(* CODESYS project CtaSysGrafanaLibPanel_1.0.0.0.library
   Description: SYS Grafana Library der CTA
   Version: 1.0.0.0
   Title: CtaSysGrafanaLibPanel
   Author: SIS
   Company: CTA
   Placeholder: CtaSysGrafanaLibPanel
   DocFormat: reStructuredText
   CompiledLibraryCompatibilityVersion: CODESYS V3.5 SP16 Patch 3
   LanguageModelAttribute: qualified-access-only
   DefaultNamespace: CtaSysGrafanaLibPanel

Project tree, tasks and I/O mapping:
  libraries: SysProcess, 3.5.17.0 (System); Standard, 3.5.18.0 (System); StringUtils, 3.5.18.0 (System); CtaVisSymbols, 1.0.0.0 (CTA); VisuSymbols, 4.5.0.0 (System); SysTypes Interfaces, * (System)
  40 Visualizations/
    visualisation VIS_GRAFANA_LIB_PANEL
    visualisation VIS_POPUP_GRAFANA
  00000000-0000-0000-0000-000000000000|D:\CoDeSys\LibrariesV3\trunk\Intern\CAA\CAA Template\3.4.0.0 draft\Placeholder.xml
  00000000-0000-0000-0000-000000000000|D:\CoDeSys\LibrariesV3\trunk\Intern\CAA\CAA Template\3.2.0.3 draft\Prefix.pdf
  00000000-0000-0000-0000-000000000000|D:\CoDeSys\LibrariesV3\trunk\Intern\CAA\CAA Template\3.5.2.0 draft\Placeholder.xml
  20 Structs/
  50 Images/
  10 Documenation/
    global variables VersionHistory
    global variables readMe
  21 Interface/
    interface ITF_GRAFANA_LIB_PANEL: TABLE_EXECUTE, TABLE_STATUS, LIB_PANEL_UID
  11 Library Parameter/
    global variables Parameter
  12 Konstanten/
  60 Textlisten/
  13 Globale Variablen/
    global variables GVL_GRAFANA_CONSTANT
    global variables GVL_GRAFANA_LIB_PANEL
  text list GlobalTextList
  5ce3da45-db07-42e7-a21c-a00fff4ed8f6|C:\Users\sis\Downloads\dip-switch.svg
  5ce3da45-db07-42e7-a21c-a00fff4ed8f6|C:\Users\sis\Downloads\lightning-bolt-circle.svg
  30 Program Organization Units/
    function block FB_GRAFANA_LIB_PANEL [ST]: TIMESERIES_HEAD, TIMESERIES_FOOTER, STATETIMELINE_HEAD, STATETIMELINE_FOOTER, GET_VERSION, UPDATE_VERSION, DO_HEADER, DO_FOOTER, DO_TEMP_FILES, DELETE_TEMP_FILES, URL, NEW_LIB_PANEL, UPDATE_LIB_PANEL, GET_LIB_PANEL, GET_API_KEY, DELETE_API_KEY, DATA, READY_FOR_DATA, FB_EXIT, FB_INIT, TABLE_STATUS, EXECUTE, LIB_PANEL_UID, TABLE_EXECUTE, REMOVE_SPECIALCHAR, CREATE_DYN_DATA, DELETE_DYN_DATA
    function fcRemoveSpezialChar [ST]
  5ce3da45-db07-42e7-a21c-a00fff4ed8f6|C:\Users\sis\Downloads\sine-wave.svg
  5ce3da45-db07-42e7-a21c-a00fff4ed8f6|C:\Users\sis\Downloads\eye.svg
  5ce3da45-db07-42e7-a21c-a00fff4ed8f6|C:\Users\sis\Downloads\lan.svg
  22 Enumeration/
    data type FB_GRAFANA_LIB_PANEL_STATUS
    data type GRAFANA_DATABASE_TYPE
    data type GRAFANA_LIB_PANEL_TYPE
*)

// 22 Enumeration/FB_GRAFANA_LIB_PANEL_STATUS
{attribute 'qualified_only'}
{attribute 'strict'}
TYPE FB_GRAFANA_LIB_PANEL_STATUS :
(
	NO_ERROR		:= -1,
	READY 			:= 0,
	GET_API_KEY		:= 1,
	DO_TMP_FILE		:= 2,
	DO_JSON_HEADER	:= 3,
	DO_JSON_DATA	:= 4,
	DO_JSON_FOOTER	:= 5,
	DO_NEW_PANEL	:= 6,
	DO_UPDATE		:= 7,
	DELETE_API_KEY	:= 8,
	DELETE_DYNMEM	:= 9
);
END_TYPE

// 22 Enumeration/GRAFANA_DATABASE_TYPE
{attribute 'qualified_only'}
{attribute 'strict'}
TYPE GRAFANA_DATABASE_TYPE :
(
	INFLUXDB := 1
);
END_TYPE

// 22 Enumeration/GRAFANA_LIB_PANEL_TYPE
{attribute 'qualified_only'}
{attribute 'strict'}
TYPE GRAFANA_LIB_PANEL_TYPE :
(
	TIMESERIES 		:= 0,
	STATETIMELINE 	:= 1
);
END_TYPE

// 10 Documenation/VersionHistory
(* 

.. image:: ../../Images/CTA_Logo.jpg
   :align: right
   :width: 15% 

**Vorlage**   


============ =========== =========== ============================================
**Date**     **Version** **Author**  **Change**
------------ ----------- ----------- --------------------------------------------
04.03.2021   0.0.0.0     SIS         Vorlage erstellt

============ =========== =========== ============================================


*)
VAR_GLOBAL
    stInfo : STRING:= '0.0.0.0, Vorlage, CTA';
END_VAR

// 10 Documenation/readMe
(*

**ReadMe**
 
|	**Empfehlung**
|
|	Die SysGrafanaLibPanel Library dient der automatischen erstellung von Grafana Library Panels. Diese können mit dem FB_GRAFANA_LIB_PANEL erstellt werden.
|	Die erstellung des Panels wird Manuell über die Visualisierung ausgelöst. 
|	Die Daten welche für das erstellen der Panel benötigt werden können über die Methode DATA abgefüllt werden. Jeder Aufruf der Methode ist ein Data field.
|  
| *Beispiel* 

+-----------------------+---------------------------------------------------------------------------------------------------------------------------------------------------------------------------------------------------------------------------------------------------------------------------------------------------------------------------------------------------------------------------------------------------------------------------------------+
| Beschreibung          |  Code                                                                                                                                                                                                                                                                                                                                                                                                                                 |
+=======================+=======================================================================================================================================================================================================================================================================================================================================================================================================================================+
| Pou oder SmFb         | .. code-block:: codesys                                                                                                                                                                                                                                                                                                                                                                                                               |
|                       |                                                                                                                                                                                                                                                                                                                                                                                                                                       |
|                       |	// Deklaration als VAR im POU oder dem selbsterstellten Funktionsbaustein                                                                                                                                                                                                                                                                                                                                                       	|
|                       |   VAR   																																																																																																								|
|						|	    (*Grafana Test Panel*)																																																		 																																																	|
|						|		fbGrafanaTestPanel  : CtaSysGrafanaLibPanel.FB_GRAFANA_LIB_PANEL;                                                                                                                                                                                                                                                                                                                                								|
| 						|	END_VAR                                                                                                                                                                                                                                                                                                                                                                                                                         	|
+-----------------------+---------------------------------------------------------------------------------------------------------------------------------------------------------------------------------------------------------------------------------------------------------------------------------------------------------------------------------------------------------------------------------------------------------------------------------------+
| Code                  | .. code-block:: codesys                                                                                                                                                                                                                                                                                                                                                                                                               |
|                       |   																																																																																																									|
| 						|																																																																																																										|
|                       |	fbGrafanaTestPanel(	LIB_PANEL_TYPE	:= GRAFANA_LIB_PANEL_TYPE.TIMESERIES,																																																																																							|
| 						|						DATABASE_TYPE	:= GRAFANA_DATABASE_TYPE.INFLUXDB,               																																																																																				|
|						|						stDATABASE_NAME	:= CtaAppTrendLog.fcGetInfluxDbName,	                             																																																																															|
|						|						stLIB_PANEL_UID := "UniqPanelName",                         																																																																																					| 
|						|						stIP			:= CtaAppTrendLog.fcGetInfluxDbIp,                                         																																																																														| 
|						|						uiPORT			:= CtaAppTrendLog.fcGetInfluxDbPort,                                              																																																																												| 
|						|						stUSER			:= 'admin',                                           																																																																																			|
|						|						stPASSWORD		:= 'CtaElektro');                                  																																																																																				| 
|						|																																																																																																										| 
|						|																										   	 																																																																															| 
|						|	IF fbGrafanaTestPanel.READY_FOR_DATA() THEN																											    																																																																			| 
|						|		fbGrafanaTestPanel.DATA("TrendLogId","Alias","BOOL?","LetztesFeld?");                       																																				    																																												| 
|						|	END_IF;																																													    																																																										| 
|						|																				    																																																																																					| 
|						|																																					    																																																																				| 
|						|																																																																																																										| 
|						|																																																																																																										| 
|						|																																																																																																										| 
+-----------------------+---------------------------------------------------------------------------------------------------------------------------------------------------------------------------------------------------------------------------------------------------------------------------------------------------------------------------------------------------------------------------------------------------------------------------------------+
*)      
VAR_GLOBAL
    xReadMeDone              :   BOOL;
END_VAR

// 13 Globale Variablen/GVL_GRAFANA_CONSTANT
{attribute 'qualified_only'}
VAR_GLOBAL CONSTANT
	MAX_SUPORTET_DATABASES	 : INT	:= 1;
	AY_GRAFANA_DATABASE_TYPE : ARRAY[1..MAX_SUPORTET_DATABASES] OF STRING	:= ['influxdb'];
END_VAR

// 13 Globale Variablen/GVL_GRAFANA_LIB_PANEL
{attribute 'qualified_only'}
VAR_GLOBAL
	AY_FB_GRAFANA_LIB_PANEL	:	ARRAY[1..Parameter.iMaxLibPanels] OF ITF_GRAFANA_LIB_PANEL;
	diMissedMemory			:	DINT;
	diNextFreePlace			:	DINT;
	iMaxShow				:	INT;
	xMemoryError			:	BOOL;
	dwSync					:	DWORD;
END_VAR

// 11 Library Parameter/Parameter
{attribute 'qualified_only'}
VAR_GLOBAL CONSTANT
    iMaxLibPanels :   INT   := 60;         // Maximale Anzahl verwendeter AT-Bausteine    
END_VAR

// 30 Program Organization Units/FB_GRAFANA_LIB_PANEL
FUNCTION_BLOCK FB_GRAFANA_LIB_PANEL IMPLEMENTS ITF_GRAFANA_LIB_PANEL
VAR_INPUT
	LIB_PANEL_TYPE	:	GRAFANA_LIB_PANEL_TYPE;
	DATABASE_TYPE	:	GRAFANA_DATABASE_TYPE;
	stDATABASE_NAME	:	STRING(40);
	stLIB_PANEL_UID	:	STRING(40);
	stIP			:	STRING(15);
	uiPORT			:	UINT;
	stUSER			:	STRING;
	stPASSWORD		:	STRING;
END_VAR
VAR_OUTPUT
	xREADY			:	BOOL;
	xBUSY			:	BOOL;
	xOK				:	BOOL	:= TRUE;
	xERROR			:	BOOL;
	ERROR_ON_STATE	:	FB_GRAFANA_LIB_PANEL_STATUS;	
END_VAR
VAR
	stLIB_PANEL_UID_NO_SPC	:	STRING;
	xExecute				:	BOOL;
	stURL					:	POINTER TO STRING(255);
	stKEY					:	POINTER TO STRING(255);
	stKEY_ID				:	POINTER TO STRING(10);
	stVersion				:	POINTER TO STRING(40);
	stResult				:	POINTER TO STRING(255);	
	stTemp					:	POINTER TO STRING(2000);
	stCommand				:	POINTER TO STRING(2000);
	RTS_IEC_RESULT			:	SysTypes.RTS_IEC_RESULT;
	STATUS					:	FB_GRAFANA_LIB_PANEL_STATUS;
	uiDataSecurity			:	UINT;
	dwTest					:	DWORD;
END_VAR

(* STATE MACHINE *)
CASE STATUS OF
	(* READY *)
	FB_GRAFANA_LIB_PANEL_STATUS.READY 			:
		xREADY	:= TRUE;
		xBUSY	:= FALSE;
		IF xExecute THEN
			xREADY			:= FALSE;
			xBUSY			:= TRUE;
			dwTest := TEST_AND_SET(GVL_GRAFANA_LIB_PANEL.dwSync);
			IF dwTest = 0 THEN
				CREATE_DYN_DATA();
				URL();	
				STATUS 			:= FB_GRAFANA_LIB_PANEL_STATUS.GET_API_KEY;					
				ERROR_ON_STATE	:= FB_GRAFANA_LIB_PANEL_STATUS.NO_ERROR;
				xOK    			:= FALSE;
				xERROR 			:= FALSE;
				xExecute		:= FALSE;
				uiDataSecurity	:= 0;
			END_IF;
		END_IF;	
	
	(* GET API KEY *)
	FB_GRAFANA_LIB_PANEL_STATUS.GET_API_KEY		:
		REMOVE_SPECIALCHAR();
		GET_API_KEY();
		IF xERROR AND ERROR_ON_STATE = FB_GRAFANA_LIB_PANEL_STATUS.NO_ERROR THEN
			ERROR_ON_STATE := FB_GRAFANA_LIB_PANEL_STATUS.GET_API_KEY;
		END_IF;
		
	(* DO TEMP FILE *)
	FB_GRAFANA_LIB_PANEL_STATUS.DO_TMP_FILE		:
		DO_TEMP_FILES();
		IF xERROR AND ERROR_ON_STATE = FB_GRAFANA_LIB_PANEL_STATUS.NO_ERROR THEN
			ERROR_ON_STATE := FB_GRAFANA_LIB_PANEL_STATUS.DO_TMP_FILE;
		END_IF;
		
	(* DO JSON HEADER *)
	FB_GRAFANA_LIB_PANEL_STATUS.DO_JSON_HEADER	:
		DO_HEADER();
		IF xERROR AND ERROR_ON_STATE = FB_GRAFANA_LIB_PANEL_STATUS.NO_ERROR THEN
			ERROR_ON_STATE := FB_GRAFANA_LIB_PANEL_STATUS.DO_JSON_HEADER;
		END_IF;
		
	(* DO JSON DATA *)
	FB_GRAFANA_LIB_PANEL_STATUS.DO_JSON_DATA		:
		(* Wait for DATA *) ;
		IF xERROR AND ERROR_ON_STATE = FB_GRAFANA_LIB_PANEL_STATUS.NO_ERROR THEN
			ERROR_ON_STATE := FB_GRAFANA_LIB_PANEL_STATUS.DO_JSON_DATA;
		END_IF;	
		
	(* DO JSON FOOTER *)	
	FB_GRAFANA_LIB_PANEL_STATUS.DO_JSON_FOOTER	:
		DO_FOOTER();
		IF xERROR AND ERROR_ON_STATE = FB_GRAFANA_LIB_PANEL_STATUS.NO_ERROR THEN
			ERROR_ON_STATE := FB_GRAFANA_LIB_PANEL_STATUS.DO_JSON_FOOTER;
		END_IF;
		
	(* DO NEW PANEL *)
	FB_GRAFANA_LIB_PANEL_STATUS.DO_NEW_PANEL		:
		NEW_LIB_PANEL();
		IF xERROR AND ERROR_ON_STATE = FB_GRAFANA_LIB_PANEL_STATUS.NO_ERROR THEN
			ERROR_ON_STATE := FB_GRAFANA_LIB_PANEL_STATUS.DO_NEW_PANEL;
		END_IF;
		
	(* DO PANEL UPDATE *)
	FB_GRAFANA_LIB_PANEL_STATUS.DO_UPDATE		:
		UPDATE_LIB_PANEL();
		IF xERROR AND ERROR_ON_STATE = FB_GRAFANA_LIB_PANEL_STATUS.NO_ERROR THEN
			ERROR_ON_STATE := FB_GRAFANA_LIB_PANEL_STATUS.DO_UPDATE;
		END_IF;
		
	(* DELETE API KEY *)
	FB_GRAFANA_LIB_PANEL_STATUS.DELETE_API_KEY	:
		DELETE_API_KEY();
		DELETE_TEMP_FILES();
		xOK 	:= NOT xERROR;
		STATUS	:= FB_GRAFANA_LIB_PANEL_STATUS.DELETE_DYNMEM;
		IF xERROR AND ERROR_ON_STATE = FB_GRAFANA_LIB_PANEL_STATUS.NO_ERROR THEN
			ERROR_ON_STATE := FB_GRAFANA_LIB_PANEL_STATUS.DELETE_API_KEY;
		END_IF;
	(* DELETE MEM *)
	FB_GRAFANA_LIB_PANEL_STATUS.DELETE_DYNMEM :
		DELETE_DYN_DATA();
		STATUS	:= FB_GRAFANA_LIB_PANEL_STATUS.READY;
		GVL_GRAFANA_LIB_PANEL.dwSync := 0;
	ELSE
		STATUS := FB_GRAFANA_LIB_PANEL_STATUS.DELETE_DYNMEM;
END_CASE

METHOD PRIVATE TIMESERIES_HEAD : BOOL
VAR_INPUT
END_VAR
IF stURL <> 0 AND stKEY <> 0 AND stKEY_ID <> 0 AND stVersion <> 0 AND stResult <> 0 AND stTemp <> 0 AND stCommand <> 0 THEN
	stCommand^ := '';
	stTemp^:= '';
	stTemp^:= 'echo $'{
	"uid": "';
	Stu.StrConcatA(pstFrom:= ADR(stTemp^),pstTo := ADR(stCommand^),TO_INT(SIZEOF(stCommand^)));
	stTemp^:= '';
	stTemp^:= stLIB_PANEL_UID_NO_SPC;
	Stu.StrConcatA(pstFrom:= ADR(stTemp^),pstTo := ADR(stCommand^),TO_INT(SIZEOF(stCommand^)));
	stTemp^ := '';
	stTemp^ := '",
	"folderId": 0,
	"name": "';
	Stu.StrConcatA(pstFrom:= ADR(stTemp^),pstTo := ADR(stCommand^),TO_INT(SIZEOF(stCommand^)));
	stTemp^:= '';
	stTemp^:= stLIB_PANEL_UID;
	Stu.StrConcatA(pstFrom:= ADR(stTemp^),pstTo := ADR(stCommand^),TO_INT(SIZEOF(stCommand^)));
	stTemp^ := '';
	stTemp^ := '",
	  "version": 1,
	  "model":
	{
	  "type": "timeseries",
	  "title": "';
	Stu.StrConcatA(pstFrom:= ADR(stTemp^),pstTo := ADR(stCommand^),TO_INT(SIZEOF(stCommand^)));
	stTemp^ := '';
	stTemp^ := stLIB_PANEL_UID;
	Stu.StrConcatA(pstFrom:= ADR(stTemp^),pstTo := ADR(stCommand^),TO_INT(SIZEOF(stCommand^)));
	stTemp^ := '';
	stTemp^ := '",
		"targets": [
		{
		  "refId": "A",
		  "datasource": {
			"type": "';
	Stu.StrConcatA(pstFrom:= ADR(stTemp^),pstTo := ADR(stCommand^),TO_INT(SIZEOF(stCommand^)));
	
	stTemp^ := '';
	IF DATABASE_TYPE >= GRAFANA_DATABASE_TYPE.INFLUXDB AND DATABASE_TYPE <= GVL_GRAFANA_CONSTANT.MAX_SUPORTET_DATABASES THEN
		stTemp^ := GVL_GRAFANA_CONSTANT.AY_GRAFANA_DATABASE_TYPE[DATABASE_TYPE];
	ELSE
		stTemp^ := GVL_GRAFANA_CONSTANT.AY_GRAFANA_DATABASE_TYPE[GRAFANA_DATABASE_TYPE.INFLUXDB];	
	END_IF;
	Stu.StrConcatA(pstFrom:= ADR(stTemp^),pstTo := ADR(stCommand^),TO_INT(SIZEOF(stCommand^)));
	
	stTemp^ := '';
	stTemp^ := '",
			"uid": ""
		  },
		  "policy": "default",
		  "resultFormat": "time_series",
		  "orderByTime": "ASC",
		  "tags": [],
		  "groupBy": [
			{
			  "type": "time",
			  "params": [
				"$$__interval"
			  ]
			},
			{
			  "type": "fill",
			  "params": [
				"none"
			  ]
			}
		  ],
		  "select": [$' > /tmp/';
	Stu.StrConcatA(pstFrom:= ADR(stTemp^),pstTo := ADR(stCommand^),TO_INT(SIZEOF(stCommand^)));
	stTemp^ := '';
	stTemp^ := stLIB_PANEL_UID_NO_SPC;
	
	Stu.StrConcatA(pstFrom:= ADR(stTemp^),pstTo := ADR(stCommand^),TO_INT(SIZEOF(stCommand^)));
	stTemp^ := '';
	stTemp^ := '.txt';
	Stu.StrConcatA(pstFrom:= ADR(stTemp^),pstTo := ADR(stCommand^),TO_INT(SIZEOF(stCommand^)));
		  
	SysProcess_Implementation.SysProcessExecuteCommand2(stCommand^,stResult^,SIZEOF(stResult^),ADR(RTS_IEC_RESULT));
	
	TIMESERIES_HEAD	:= RTS_IEC_RESULT = 0;
ELSE
	STATUS := FB_GRAFANA_LIB_PANEL_STATUS.DELETE_DYNMEM;
END_IF;
END_METHOD

METHOD PRIVATE TIMESERIES_FOOTER : BOOL;
VAR_INPUT
END_VAR
IF stURL <> 0 AND stKEY <> 0 AND stKEY_ID <> 0 AND stVersion <> 0 AND stResult <> 0 AND stTemp <> 0 AND stCommand <> 0 THEN
	stCommand^ := '';
	stCommand^ := 'echo $'],
				  "measurement": "';
	stTemp^ := '';
	stTemp^ := stDATABASE_NAME;
	
	Stu.StrConcatA(pstFrom:= ADR(stTemp^),pstTo := ADR(stCommand^),TO_INT(SIZEOF(stCommand^)));
	
	stTemp^ := '';
	stTemp^ := '",
				  "alias": "$$col"
					}
					  ],
					  "options": {
						"tooltip": {
						  "mode": "multi"
						},
						"legend": {
						  "displayMode": "table",
						  "placement": "bottom",
						  "calcs": []
						}
					  },
					  "fieldConfig": {
						"defaults": {
						  "custom": {
							"drawStyle": "line",
							"lineInterpolation": "smooth",
							"barAlignment": 0,
							"lineWidth": 1,
							"fillOpacity": 0,
							"gradientMode": "none",
							"spanNulls": false,
							"showPoints": "auto",
							"pointSize": 5,
							"stacking": {
							  "mode": "none",
							  "group": "A"
							},
							"axisPlacement": "auto",
							"axisLabel": "",
							"scaleDistribution": {
							  "type": "linear"
							},
							"hideFrom": {
							  "tooltip": false,
							  "viz": false,
							  "legend": false
							},
							"thresholdsStyle": {
							  "mode": "off"
							}
						  },
						  "color": {
							"mode": "palette-classic"
						  },
						  "thresholds": {
							"mode": "absolute",
							"steps": [
							  {
								"color": "green",
								"value": null
							  }
							]
						  },
						  "mappings": []
						},
						"overrides": []
					  },
					  "datasource": null
					},
			  "kind": 1
			}$' >> /tmp/';
	Stu.StrConcatA(pstFrom:= ADR(stTemp^),pstTo := ADR(stCommand^),TO_INT(SIZEOF(stCommand^)));
	
	stTemp^ := '';
	stTemp^ := stLIB_PANEL_UID_NO_SPC;
	
	Stu.StrConcatA(pstFrom:= ADR(stTemp^),pstTo := ADR(stCommand^),TO_INT(SIZEOF(stCommand^)));
	stTemp^ := '';
	stTemp^ := '.txt';		
	Stu.StrConcatA(pstFrom:= ADR(stTemp^),pstTo := ADR(stCommand^),TO_INT(SIZEOF(stCommand^)));
	
	SysProcess_Implementation.SysProcessExecuteCommand2(stCommand^,stResult^,SIZEOF(stResult^),ADR(RTS_IEC_RESULT));
	
	TIMESERIES_FOOTER	:= RTS_IEC_RESULT = 0;
ELSE
	STATUS := FB_GRAFANA_LIB_PANEL_STATUS.DELETE_DYNMEM;
END_IF;
END_METHOD

METHOD PRIVATE STATETIMELINE_HEAD : BOOL
VAR_INPUT
END_VAR
IF stURL <> 0 AND stKEY <> 0 AND stKEY_ID <> 0 AND stVersion <> 0 AND stResult <> 0 AND stTemp <> 0 AND stCommand <> 0 THEN
	stCommand^ := '';
	stTemp^:= '';
	stTemp^:= 'echo $'{
	"uid": "';
	Stu.StrConcatA(pstFrom:= ADR(stTemp^),pstTo := ADR(stCommand^),TO_INT(SIZEOF(stCommand^)));
	stTemp^:= '';
	stTemp^:= stLIB_PANEL_UID_NO_SPC;
	Stu.StrConcatA(pstFrom:= ADR(stTemp^),pstTo := ADR(stCommand^),TO_INT(SIZEOF(stCommand^)));
	stTemp^ := '';
	stTemp^ := '",
	"folderId": 0,
	"name": "';
	Stu.StrConcatA(pstFrom:= ADR(stTemp^),pstTo := ADR(stCommand^),TO_INT(SIZEOF(stCommand^)));
	stTemp^:= '';
	stTemp^:= stLIB_PANEL_UID;
	Stu.StrConcatA(pstFrom:= ADR(stTemp^),pstTo := ADR(stCommand^),TO_INT(SIZEOF(stCommand^)));
	stTemp^ := '';
	stTemp^ := '",
	  "version": 1,
	  "model":
	{
	  "type": "state-timeline",
	  "title": "';
	Stu.StrConcatA(pstFrom:= ADR(stTemp^),pstTo := ADR(stCommand^),TO_INT(SIZEOF(stCommand^)));
	stTemp^ := '';
	stTemp^ := stLIB_PANEL_UID;
	Stu.StrConcatA(pstFrom:= ADR(stTemp^),pstTo := ADR(stCommand^),TO_INT(SIZEOF(stCommand^)));
	stTemp^ := '';
	stTemp^ := '",
	  "fieldConfig": {
		"defaults": {
		  "custom": {
			"lineWidth": 0,
			"fillOpacity": 70
		  },
		  "color": {
			"mode": "fixed"
		  },
		  "thresholds": {
			"mode": "absolute",
			"steps": [
			  {
				"color": "green",
				"value": null
			  }
			]
		  },
		  "mappings": []
		},
		"overrides": []
	  },
	  "options": {
		"mergeValues": true,
		"showValue": "auto",
		"alignValue": "left",
		"rowHeight": 0.9,
		"legend": {
		  "displayMode": "hidden",
		  "placement": "bottom"
		},
		"tooltip": {
		  "mode": "single"
		}
	  },
	  "targets": [
		{
		  "datasource": {
			"type": "';
	
	Stu.StrConcatA(pstFrom:= ADR(stTemp^),pstTo := ADR(stCommand^),TO_INT(SIZEOF(stCommand^)));
			
	stTemp^ := '';
	IF DATABASE_TYPE >= GRAFANA_DATABASE_TYPE.INFLUXDB AND DATABASE_TYPE <= GVL_GRAFANA_CONSTANT.MAX_SUPORTET_DATABASES THEN
		stTemp^ := GVL_GRAFANA_CONSTANT.AY_GRAFANA_DATABASE_TYPE[DATABASE_TYPE];
	ELSE
		stTemp^ := GVL_GRAFANA_CONSTANT.AY_GRAFANA_DATABASE_TYPE[GRAFANA_DATABASE_TYPE.INFLUXDB];	
	END_IF;
	Stu.StrConcatA(pstFrom:= ADR(stTemp^),pstTo := ADR(stCommand^),TO_INT(SIZEOF(stCommand^)));
	
	stTemp^ := '';
	stTemp^ := '",
			"uid": ""
		  },
		  "groupBy": [
			{
			  "params": [
				"$$__interval"
			  ],
			  "type": "time"
			},
			{
			  "params": [
				"none"
			  ],
			  "type": "fill"
			}
		  ],
		  "measurement": "';
	
	Stu.StrConcatA(pstFrom:= ADR(stTemp^),pstTo := ADR(stCommand^),TO_INT(SIZEOF(stCommand^)));
	
	stTemp^ := '';
	stTemp^ := stDATABASE_NAME;
	
	Stu.StrConcatA(pstFrom:= ADR(stTemp^),pstTo := ADR(stCommand^),TO_INT(SIZEOF(stCommand^)));
	
	stTemp^ := '';
	stTemp^ := '",
		  "orderByTime": "ASC",
		  "policy": "default",
		  "refId": "A",
		  "resultFormat": "time_series",
		  "select": [$' > /tmp/';
	Stu.StrConcatA(pstFrom:= ADR(stTemp^),pstTo := ADR(stCommand^),TO_INT(SIZEOF(stCommand^)));
	stTemp^ := '';
	stTemp^ := stLIB_PANEL_UID_NO_SPC;
	
	Stu.StrConcatA(pstFrom:= ADR(stTemp^),pstTo := ADR(stCommand^),TO_INT(SIZEOF(stCommand^)));
	stTemp^ := '';
	stTemp^ := '.txt';
	Stu.StrConcatA(pstFrom:= ADR(stTemp^),pstTo := ADR(stCommand^),TO_INT(SIZEOF(stCommand^)));
		  
	SysProcess_Implementation.SysProcessExecuteCommand2(stCommand^,stResult^,SIZEOF(stResult^),ADR(RTS_IEC_RESULT));
	
	STATETIMELINE_HEAD	:= RTS_IEC_RESULT = 0;
ELSE
	STATUS := FB_GRAFANA_LIB_PANEL_STATUS.DELETE_DYNMEM;
END_IF;
END_METHOD

METHOD PRIVATE STATETIMELINE_FOOTER : BOOL
VAR_INPUT
END_VAR
IF stURL <> 0 AND stKEY <> 0 AND stKEY_ID <> 0 AND stVersion <> 0 AND stResult <> 0 AND stTemp <> 0 AND stCommand <> 0 THEN
	stCommand^ := '';
	stCommand^ := 'echo $'],
				  "tags": [],
				  "alias": "$$col"
				}
			  ],
			  "id": 0,
			  "datasource": null
			},
			  "kind": 1
			}$' >> /tmp/';
	
	stTemp^ := '';
	stTemp^ := stLIB_PANEL_UID_NO_SPC;
	
	Stu.StrConcatA(pstFrom:= ADR(stTemp^),pstTo := ADR(stCommand^),TO_INT(SIZEOF(stCommand^)));
	stTemp^ := '';
	stTemp^ := '.txt';		
	Stu.StrConcatA(pstFrom:= ADR(stTemp^),pstTo := ADR(stCommand^),TO_INT(SIZEOF(stCommand^)));
	
	SysProcess_Implementation.SysProcessExecuteCommand2(stCommand^,stResult^,SIZEOF(stResult^),ADR(RTS_IEC_RESULT));
	
	STATETIMELINE_FOOTER	:= RTS_IEC_RESULT = 0;
ELSE
	STATUS := FB_GRAFANA_LIB_PANEL_STATUS.DELETE_DYNMEM;
END_IF;
END_METHOD

METHOD PRIVATE GET_VERSION : BOOL
VAR_INPUT
END_VAR
IF stURL <> 0 AND stKEY <> 0 AND stKEY_ID <> 0 AND stVersion <> 0 AND stResult <> 0 AND stTemp <> 0 AND stCommand <> 0 THEN
	(* Get Version *)
	stCommand^ := '';
	stCommand^ := Standard.CONCAT(Standard.CONCAT('grep -oE $'.{0,1}version.{0,5}[0-9]$' /tmp/',stLIB_PANEL_UID_NO_SPC),'_V.txt | tail -1');
	SysProcess_Implementation.SysProcessExecuteCommand2(stCommand^,stResult^,SIZEOF(stResult^),ADR(RTS_IEC_RESULT));
	
	IF FIND(stResult^,'$N') > 1 AND FIND(stResult^,'"version"') > 0 AND RTS_IEC_RESULT = 0 THEN
		stVersion^ 	:= '';
		stVersion^ 	:= Standard.LEFT(stResult^,FIND(stResult^,'$N')-1);
		GET_VERSION := TRUE;
	ELSE
		xERROR		:= TRUE;
	END_IF;
ELSE
	STATUS := FB_GRAFANA_LIB_PANEL_STATUS.DELETE_DYNMEM;
END_IF;
END_METHOD

METHOD PRIVATE UPDATE_VERSION : BOOL
VAR_INPUT
END_VAR
IF stURL <> 0 AND stKEY <> 0 AND stKEY_ID <> 0 AND stVersion <> 0 AND stResult <> 0 AND stTemp <> 0 AND stCommand <> 0 THEN
	(* Update Version *)
	stCommand^ := '';
	stCommand^ := Standard.CONCAT(Standard.CONCAT(Standard.CONCAT(Standard.CONCAT('sed -i $'s/"version": 1/',stVersion^),'/$' /tmp/'),stLIB_PANEL_UID_NO_SPC),'.txt');
	SysProcess_Implementation.SysProcessExecuteCommand2(stCommand^,stResult^,SIZEOF(stResult),ADR(RTS_IEC_RESULT));
	
	UPDATE_VERSION := RTS_IEC_RESULT = 0;
ELSE
	STATUS := FB_GRAFANA_LIB_PANEL_STATUS.DELETE_DYNMEM;
END_IF;
END_METHOD

METHOD PRIVATE DO_HEADER : BOOL
VAR_INPUT
END_VAR
IF LIB_PANEL_TYPE = GRAFANA_LIB_PANEL_TYPE.TIMESERIES THEN
	IF TIMESERIES_HEAD()	THEN
		STATUS := FB_GRAFANA_LIB_PANEL_STATUS.DO_JSON_DATA;
	ELSE
		STATUS 	:= FB_GRAFANA_LIB_PANEL_STATUS.DELETE_API_KEY;
		xERROR	:= TRUE;
	END_IF;		
ELSIF LIB_PANEL_TYPE = GRAFANA_LIB_PANEL_TYPE.STATETIMELINE THEN
	IF STATETIMELINE_HEAD() THEN
		STATUS := FB_GRAFANA_LIB_PANEL_STATUS.DO_JSON_DATA;
	ELSE
		STATUS 	:= FB_GRAFANA_LIB_PANEL_STATUS.DELETE_API_KEY;
		xERROR	:= TRUE;
	END_IF;
ELSE
	STATUS 	:= FB_GRAFANA_LIB_PANEL_STATUS.DELETE_API_KEY;
	xERROR	:= TRUE;
END_IF;
END_METHOD

METHOD PRIVATE DO_FOOTER : BOOL
VAR_INPUT
END_VAR
IF LIB_PANEL_TYPE = GRAFANA_LIB_PANEL_TYPE.TIMESERIES THEN
	IF TIMESERIES_FOOTER()	THEN
		STATUS 	:= FB_GRAFANA_LIB_PANEL_STATUS.DO_NEW_PANEL;
	ELSE
		STATUS 	:= FB_GRAFANA_LIB_PANEL_STATUS.DELETE_API_KEY;
		xERROR	:= TRUE;
	END_IF;		
ELSIF LIB_PANEL_TYPE = GRAFANA_LIB_PANEL_TYPE.STATETIMELINE THEN
	IF STATETIMELINE_FOOTER() THEN
		STATUS := FB_GRAFANA_LIB_PANEL_STATUS.DO_NEW_PANEL;
	ELSE
		STATUS 	:= FB_GRAFANA_LIB_PANEL_STATUS.DELETE_API_KEY;
		xERROR	:= TRUE;
	END_IF;
ELSE
	STATUS 	:= FB_GRAFANA_LIB_PANEL_STATUS.DELETE_API_KEY;
	xERROR	:= TRUE;
END_IF;
END_METHOD

METHOD PRIVATE DO_TEMP_FILES : BOOL
VAR_INPUT
END_VAR
IF stURL <> 0 AND stKEY <> 0 AND stKEY_ID <> 0 AND stVersion <> 0 AND stResult <> 0 AND stTemp <> 0 AND stCommand <> 0 THEN
	(* TEMP JSON FILE *)
	stCommand^ := 	Standard.CONCAT(
					Standard.CONCAT(
										'touch /tmp/',
										stLIB_PANEL_UID_NO_SPC),
										'.txt');
	SysProcess_Implementation.SysProcessExecuteCommand2(stCommand^,stResult^,SIZEOF(stResult^),ADR(RTS_IEC_RESULT));
	
	(* TEMP JSON VERSION FILE *)
	IF RTS_IEC_RESULT = 0 THEN
		stCommand^ := 	Standard.CONCAT(
						Standard.CONCAT(
											'touch /tmp/',
											stLIB_PANEL_UID_NO_SPC),
											'_V.txt');
		SysProcess_Implementation.SysProcessExecuteCommand2(stCommand^,stResult^,SIZEOF(stResult^),ADR(RTS_IEC_RESULT));
	END_IF;
	IF RTS_IEC_RESULT = 0 THEN
		DO_TEMP_FILES 	:= TRUE;
		STATUS 		:= FB_GRAFANA_LIB_PANEL_STATUS.DO_JSON_HEADER;
	ELSE
		DO_TEMP_FILES 	:= FALSE;
		STATUS 		:= FB_GRAFANA_LIB_PANEL_STATUS.DELETE_API_KEY;	
		xERROR		:= TRUE;
	END_IF;
ELSE
	STATUS := FB_GRAFANA_LIB_PANEL_STATUS.DELETE_DYNMEM;
END_IF;
END_METHOD

METHOD PRIVATE DELETE_TEMP_FILES : BOOL
VAR_INPUT
END_VAR
IF stURL <> 0 AND stKEY <> 0 AND stKEY_ID <> 0 AND stVersion <> 0 AND stResult <> 0 AND stTemp <> 0 AND stCommand <> 0 THEN
	(* TEMP JSON FILE *)
	stCommand^ := 	Standard.CONCAT(
					Standard.CONCAT(
										'rm /tmp/',
										stLIB_PANEL_UID_NO_SPC),
										'.txt');
	SysProcess_Implementation.SysProcessExecuteCommand2(stCommand^,stResult^,SIZEOF(stResult),ADR(RTS_IEC_RESULT));
	
	(* TEMP JSON VERSION FILE *)
	stCommand^ := 	Standard.CONCAT(
					Standard.CONCAT(
										'rm /tmp/',
										stLIB_PANEL_UID_NO_SPC),
										'_V.txt');
	SysProcess_Implementation.SysProcessExecuteCommand2(stCommand^,stResult^,SIZEOF(stResult^),ADR(RTS_IEC_RESULT));
	
	IF RTS_IEC_RESULT <> 0 THEN
		xERROR := TRUE;
	END_IF;
ELSE
	STATUS := FB_GRAFANA_LIB_PANEL_STATUS.DELETE_DYNMEM;
END_IF;
END_METHOD

METHOD URL : BOOL
VAR_INPUT
END_VAR
IF stURL <> 0 AND stKEY <> 0 AND stKEY_ID <> 0 AND stVersion <> 0 AND stResult <> 0 AND stTemp <> 0 AND stCommand <> 0 THEN
	(* GET URL *)
	stURL^ := '';
	stURL^ := 		Standard.CONCAT	(
					Standard.CONCAT	(
					Standard.CONCAT	(
					Standard.CONCAT	(
					Standard.CONCAT	(
					Standard.CONCAT	(
					Standard.CONCAT	(
										'https://',
										stUSER),
										':'),
										stPASSWORD),
										'@'),
										stIP),
										':'),
										TO_STRING(uiPORT));
ELSE
	STATUS := FB_GRAFANA_LIB_PANEL_STATUS.DELETE_DYNMEM;
END_IF;
END_METHOD

METHOD PRIVATE NEW_LIB_PANEL : BOOL
VAR_INPUT
END_VAR
IF stURL <> 0 AND stKEY <> 0 AND stKEY_ID <> 0 AND stVersion <> 0 AND stResult <> 0 AND stTemp <> 0 AND stCommand <> 0 THEN
	(* Create Panel *)
	stCommand^ := '';
	stTemp^:= '';
	stTemp^:= 'curl -X POST ';
	Stu.StrConcatA(pstFrom:= ADR(stTemp^),pstTo := ADR(stCommand^),TO_INT(SIZEOF(stCommand^)));
	Stu.StrConcatA(pstFrom:= ADR(stUrl^),pstTo := ADR(stCommand^),TO_INT(SIZEOF(stCommand^)));
	stTemp^:= '';
	stTemp^:= '/api/library-elements --insecure -H "Accept: application/json" -H "Content-Type: application/json" -H "Authorization: Bearer ';
	Stu.StrConcatA(pstFrom:= ADR(stTemp^),pstTo := ADR(stCommand^),TO_INT(SIZEOF(stCommand^)));
	Stu.StrConcatA(pstFrom:= ADR(stKey^),pstTo := ADR(stCommand^),TO_INT(SIZEOF(stCommand^)));
	stTemp^:= '';
	stTemp^:= Standard.CONCAT(Standard.CONCAT('" -d @/tmp/',stLIB_PANEL_UID_NO_SPC),'.txt');
	Stu.StrConcatA(pstFrom:= ADR(stTemp^),pstTo := ADR(stCommand^),TO_INT(SIZEOF(stCommand^)));
	SysProcess_Implementation.SysProcessExecuteCommand2(stCommand^,stResult^,SIZEOF(stResult^),ADR(RTS_IEC_RESULT));
	
	IF Standard.FIND(stResult^,'{"result":{"id":') > 0 AND RTS_IEC_RESULT = 0 THEN
		NEW_LIB_PANEL := TRUE;
		STATUS 		  := FB_GRAFANA_LIB_PANEL_STATUS.DELETE_API_KEY;
	ELSE
		NEW_LIB_PANEL := FALSE;
		STATUS 		  := FB_GRAFANA_LIB_PANEL_STATUS.DO_UPDATE;	
	END_IF;
ELSE
	STATUS := FB_GRAFANA_LIB_PANEL_STATUS.DELETE_DYNMEM;
END_IF;
END_METHOD

METHOD PRIVATE UPDATE_LIB_PANEL : BOOL
VAR_INPUT
END_VAR
IF stURL <> 0 AND stKEY <> 0 AND stKEY_ID <> 0 AND stVersion <> 0 AND stResult <> 0 AND stTemp <> 0 AND stCommand <> 0 THEN
	(* Update Panel *)
	IF GET_LIB_PANEL() THEN
		IF GET_VERSION() THEN
			IF UPDATE_VERSION() THEN
				stCommand^ := '';
				stTemp^:= '';
				stTemp^:= 'curl -X PATCH ';
				Stu.StrConcatA(pstFrom:= ADR(stTemp^),pstTo := ADR(stCommand^),TO_INT(SIZEOF(stCommand^)));
				Stu.StrConcatA(pstFrom:= ADR(stUrl^),pstTo := ADR(stCommand^),TO_INT(SIZEOF(stCommand^)));
				stTemp^:= '';
				stTemp^:= Standard.CONCAT(Standard.CONCAT('/api/library-elements/',stLIB_PANEL_UID_NO_SPC),' --insecure -H "Accept: application/json" -H "Content-Type: application/json" -H "Authorization: Bearer ');
				Stu.StrConcatA(pstFrom:= ADR(stTemp^),pstTo := ADR(stCommand^),TO_INT(SIZEOF(stCommand^)));
				Stu.StrConcatA(pstFrom:= ADR(stKey^),pstTo := ADR(stCommand^),TO_INT(SIZEOF(stCommand^)));
				stTemp^:= '';
				stTemp^:= Standard.CONCAT(Standard.CONCAT('" -d @/tmp/',stLIB_PANEL_UID_NO_SPC),'.txt');
				Stu.StrConcatA(pstFrom:= ADR(stTemp^),pstTo := ADR(stCommand^),TO_INT(SIZEOF(stCommand^)));
				SysProcess_Implementation.SysProcessExecuteCommand2(stCommand^,stResult^,SIZEOF(stResult^),ADR(RTS_IEC_RESULT));
				
				IF Standard.FIND(stResult^,'{"result":{"id":') > 0 AND RTS_IEC_RESULT = 0 THEN
					UPDATE_LIB_PANEL := TRUE;
				ELSE
					xERROR	:= TRUE;
				END_IF;
			END_IF;
		END_IF;
	END_IF;
	STATUS := FB_GRAFANA_LIB_PANEL_STATUS.DELETE_API_KEY;
ELSE
	STATUS := FB_GRAFANA_LIB_PANEL_STATUS.DELETE_DYNMEM;
END_IF;
END_METHOD

METHOD PRIVATE GET_LIB_PANEL : BOOL
VAR_INPUT
END_VAR
IF stURL <> 0 AND stKEY <> 0 AND stKEY_ID <> 0 AND stVersion <> 0 AND stResult <> 0 AND stTemp <> 0 AND stCommand <> 0 THEN
	(* Get LIB PANEL FROM GRAFANA *)
	stCommand^	:= '';
	stTemp^		:= '';
	stTemp^		:= 'curl -X GET ';
	Stu.StrConcatA(pstFrom:= ADR(stTemp^),pstTo := ADR(stCommand^),TO_INT(SIZEOF(stCommand^)));
	Stu.StrConcatA(pstFrom:= ADR(stURL^),pstTo := ADR(stCommand^),TO_INT(SIZEOF(stCommand^)));
	stTemp^:= '';
	stTemp^:= Standard.CONCAT(Standard.CONCAT('/api/library-elements/',stLIB_PANEL_UID_NO_SPC),' --insecure -H "Accept: application/json" -H "Content-Type: application/json" -H "Authorization: Bearer ');
	Stu.StrConcatA(pstFrom:= ADR(stTemp^),pstTo := ADR(stCommand^),TO_INT(SIZEOF(stCommand^)));
	Stu.StrConcatA(pstFrom:= ADR(stKEY^),pstTo := ADR(stCommand^),TO_INT(SIZEOF(stCommand^)));
	stTemp^:= '';
	stTemp^:= Standard.CONCAT(Standard.CONCAT('" > /tmp/',stLIB_PANEL_UID_NO_SPC),'_V.txt');
	Stu.StrConcatA(pstFrom:= ADR(stTemp^),pstTo := ADR(stCommand^),TO_INT(SIZEOF(stCommand^)));
	SysProcess_Implementation.SysProcessExecuteCommand2(stCommand^,stResult^,SIZEOF(stResult^),ADR(RTS_IEC_RESULT));
	
	GET_LIB_PANEL := RTS_IEC_RESULT = 0;
ELSE
	STATUS := FB_GRAFANA_LIB_PANEL_STATUS.DELETE_DYNMEM;
END_IF;
END_METHOD

METHOD PRIVATE GET_API_KEY : BOOL
VAR
	iPos1		:	INT;
	ipos2		:	INT;
END_VAR
IF stURL <> 0 AND stKEY <> 0 AND stKEY_ID <> 0 AND stVersion <> 0 AND stResult <> 0 AND stTemp <> 0 AND stCommand <> 0 THEN
	stTemp^		:= '';
	stCommand^	:= '';
	(*GET API KEY*)	
	stCommand^:= 	Standard.CONCAT	(
					Standard.CONCAT	(
					Standard.CONCAT	(
					Standard.CONCAT	(
										'curl -X POST --insecure -H "Content-Type: application/json" -d $'{"name": "',
										stLIB_PANEL_UID_NO_SPC),
										'Key", "role": "Admin"}$' '),
										stURL^),
										'/api/auth/keys');
		
	// Bsp 'curl -X POST --insecure -H "Content-Type: application/json" -d $'{"name":"CtaKey", "role": "Admin"}$' https://admin:CtaElektro@10.0.1.12:3000/api/auth/keys';
	
	SysProcess_Implementation.SysProcessExecuteCommand2(stCommand^,stResult^,SIZEOF(stResult^),ADR(RTS_IEC_RESULT));
	IF Standard.FIND(stResult^,'"key":"') > 0 AND RTS_IEC_RESULT = 0 THEN
		iPos2 		:= Standard.FIND(stResult^,'"key":"')+Standard.LEN('"key":"');
		ipos1 		:= LEN(stResult^)-(Standard.FIND(stResult^,'"key":"')+Standard.LEN('"key":"'))-1;
		stKey^ 		:= Standard.MID(stResult^,iPos1,ipos2);
		stKEY_ID^  	:= Standard.MID(stResult^,FIND(stResult^,',"name":')-(FIND(stResult^,'"id":')+LEN('"id":')),FIND(stResult^,'"id":')+LEN('"id":'));
		GET_API_KEY := TRUE;
		STATUS		:= FB_GRAFANA_LIB_PANEL_STATUS.DO_TMP_FILE;
	ELSE
		STATUS		:= FB_GRAFANA_LIB_PANEL_STATUS.DELETE_API_KEY;
		xERROR		:= TRUE;
	END_IF;
ELSE
	STATUS := FB_GRAFANA_LIB_PANEL_STATUS.DELETE_DYNMEM;
END_IF;
END_METHOD

METHOD PRIVATE DELETE_API_KEY
VAR_INPUT
END_VAR
IF stURL <> 0 AND stKEY <> 0 AND stKEY_ID <> 0 AND stVersion <> 0 AND stResult <> 0 AND stTemp <> 0 AND stCommand <> 0 THEN
	stCommand^ := 	Standard.CONCAT(
					Standard.CONCAT(
					Standard.CONCAT(
									'curl -X DELETE --insecure ',
									stURL^),
									'/api/auth/keys/'),stKEY_ID^);
		
	SysProcess_Implementation.SysProcessExecuteCommand2(stCommand^,stResult^,SIZEOF(stResult^),ADR(RTS_IEC_RESULT));
	
	IF RTS_IEC_RESULT <> 0 THEN
		xERROR := TRUE;
	END_IF;
ELSE
	STATUS := FB_GRAFANA_LIB_PANEL_STATUS.DELETE_DYNMEM;
END_IF;
END_METHOD

METHOD DATA : BOOL
VAR_INPUT
	stLogId			:	STRING(100);
	stAlias			:	STRING(100);
	xIsBool 		:	BOOL;	
	xIsLastField	:	BOOL;	
END_VAR         	
VAR
	uiCount 		: 	UINT;
END_VAR
IF stURL <> 0 AND stKEY <> 0 AND stKEY_ID <> 0 AND stVersion <> 0 AND stResult <> 0 AND stTemp <> 0 AND stCommand <> 0 THEN
	IF STATUS = FB_GRAFANA_LIB_PANEL_STATUS.DO_JSON_DATA THEN	
		IF stLogId <> '' OR xIsLastField THEN
			(* Create Field DATA*)
			stCommand^ := '';
			stCommand^ := 	Standard.CONCAT(
							Standard.CONCAT(
							Standard.CONCAT(
							Standard.CONCAT(
							Standard.CONCAT(
							Standard.CONCAT(
							Standard.CONCAT(
							Standard.CONCAT(					
							Standard.CONCAT(
							Standard.CONCAT(
							Standard.CONCAT(
							Standard.CONCAT(
							Standard.CONCAT(
							Standard.CONCAT(	
							Standard.CONCAT(
							Standard.CONCAT(
							Standard.CONCAT(				
							Standard.CONCAT(
							Standard.CONCAT(
							Standard.CONCAT(
							Standard.CONCAT(					
							Standard.CONCAT(
							Standard.CONCAT(
							Standard.CONCAT(
											'echo $'',	
												'['),
													'{'),
														'"type": "field",'),
														'"params": ['),
															'"'),stLogId),
														'"]'),
													'},'),
													'{'),
														'"type": "'),SEL(xIsBool,'mode",','first",')),
														'"params": []'),
													'},'),	
													'{'),
														'"type": "alias",'),
														'"params": ['),
															'"'),stAlias),
														'"]'),
													'}'),									
												SEL(xIsLastField,'],',']')),
												'$' >> /tmp/'),
												stLIB_PANEL_UID_NO_SPC),
												 '.txt');
												 
			SysProcess_Implementation.SysProcessExecuteCommand2(stCommand^,stResult^,SIZEOF(stResult^),ADR(RTS_IEC_RESULT));	
		END_IF;
		DATA			:= RTS_IEC_RESULT = 0;
		uiDataSecurity 	:= uiDataSecurity + 1;
		IF RTS_IEC_RESULT <> 0 OR uiDataSecurity >= 2000 THEN
			STATUS := FB_GRAFANA_LIB_PANEL_STATUS.DELETE_API_KEY;
			xERROR := TRUE;
		ELSIF xIsLastField THEN
			STATUS := FB_GRAFANA_LIB_PANEL_STATUS.DO_JSON_FOOTER;	
		END_IF;
	END_IF;
ELSE
	STATUS := FB_GRAFANA_LIB_PANEL_STATUS.DELETE_DYNMEM;
END_IF;
END_METHOD

METHOD READY_FOR_DATA : BOOL
READY_FOR_DATA := STATUS = FB_GRAFANA_LIB_PANEL_STATUS.DO_JSON_DATA;
END_METHOD

//FB_Exit muss explizit implementiert werden. Wenn es eine Implementierung gibt, dann wird 
//die Methode aufgerufen, bevor die Steuerung den Code der Funktionsbaustein-Instanz entfernt
//(impliziter Aufruf. Der Rückgabewert wird nicht ausgewertet.
METHOD FB_Exit: BOOL
VAR_INPUT    
bInCopyCode: BOOL;  // TRUE: Die Exit-Methode wird aufgerufen, um die Instanz zu verlassen, die hinterher kopiert wird Online-Change).  
END_VAR
DELETE_API_KEY();
DELETE_TEMP_FILES();
END_METHOD

//FB_Init ist immer implizit verfügbar und wird primär für die Initialisierung verwendet.
//Der Rückgabewert wird nicht ausgewertet. Für gezielte Einflussnahme können Sie
//die Methoden explizit deklarieren und darin mit dem Standard-Initialisierungscode 
//zusätzlichen Code bereitstellen. Sie können den Rückgabewert auswerten.
METHOD FB_Init: BOOL
VAR_INPUT    
bInitRetains: BOOL; // TRUE: Die Retain-Variablen werden initialisiert (Reset warm / Reset kalt)    
bInCopyCode: BOOL;  // TRUE: Die Instanz wird danach in den Kopiercode kopiert (Online-Change)
END_VAR
VAR
    diTempMissedMemory  :   DINT;
	diSlotId			:	DINT;
END_VAR
IF NOT bInCopyCode THEN
    IF GVL_GRAFANA_LIB_PANEL.diNextFreePlace <= UPPER_BOUND(GVL_GRAFANA_LIB_PANEL.AY_FB_GRAFANA_LIB_PANEL,1) THEN
        IF GVL_GRAFANA_LIB_PANEL.diNextFreePlace = 0 THEN
            diSlotId := __XADD(ADR(GVL_GRAFANA_LIB_PANEL.diNextFreePlace),2);
			IF diSlotId = 0 THEN
            	diSlotId := 1;
			END_IF;		
        ELSE
            diSlotId := __XADD(ADR(GVL_GRAFANA_LIB_PANEL.diNextFreePlace),1);
		END_IF;
		GVL_GRAFANA_LIB_PANEL.AY_FB_GRAFANA_LIB_PANEL[diSlotId] := THIS^;
		GVL_GRAFANA_LIB_PANEL.iMaxShow := TO_INT(GVL_GRAFANA_LIB_PANEL.diNextFreePlace -1);
    ELSE
        GVL_GRAFANA_LIB_PANEL.xMemoryError   := TRUE;
        diTempMissedMemory          := __XADD(ADR(GVL_GRAFANA_LIB_PANEL.diMissedMemory),1);
	END_IF;
END_IF;
END_METHOD

PROPERTY TABLE_STATUS : STRING
GET
IF xERROR THEN
	TABLE_STATUS	:='CtaVisSymbols.ImagePool.CtaError';	
ELSIF xBUSY THEN
	TABLE_STATUS	:='CtaVisSymbols.ImagePool.Hourglass';	
ELSIF xOK	THEN
	TABLE_STATUS	:='CtaVisSymbols.ImagePool.check_green';	
ELSE
	TABLE_STATUS	:='CtaVisSymbols.ImagePool.Hourglass';	
END_IF;
END_GET
END_PROPERTY

METHOD EXECUTE
xExecute := STATUS = FB_GRAFANA_LIB_PANEL_STATUS.READY;
END_METHOD

PROPERTY LIB_PANEL_UID : STRING
GET
LIB_PANEL_UID := stLIB_PANEL_UID;
END_GET
END_PROPERTY

PROPERTY TABLE_EXECUTE : BOOL
SET
IF TABLE_EXECUTE THEN
	EXECUTE();
END_IF;
END_SET
GET
TABLE_EXECUTE := xBUSY;
END_GET
END_PROPERTY

METHOD REMOVE_SPECIALCHAR
VAR_INPUT
END_VAR
VAR 
	uiCount : UINT;
END_VAR;
stLIB_PANEL_UID_NO_SPC := stLIB_PANEL_UID;
(* Remove ä ö ü from stLIB_PANEL_UID *)
IF stLIB_PANEL_UID_NO_SPC <> '' THEN
	stLIB_PANEL_UID_NO_SPC := fcRemoveSpezialChar(stLIB_PANEL_UID_NO_SPC);	
END_IF;
(* Remove ä ö ü from stLogId *)
IF stDATABASE_NAME <> '' THEN
	stDATABASE_NAME := fcRemoveSpezialChar(stDATABASE_NAME);	
END_IF;
END_METHOD

METHOD CREATE_DYN_DATA
VAR_INPUT
END_VAR
stURL				:=	__NEW(STRING(255));
stKEY				:=	__NEW(STRING(255));
stKEY_ID			:=	__NEW(STRING(10));
stVersion			:=	__NEW(STRING(40));
stResult			:=	__NEW(STRING(255));	
stTemp				:=	__NEW(STRING(2000));
stCommand			:=	__NEW(STRING(2000));
END_METHOD

METHOD DELETE_DYN_DATA : BOOL
VAR_INPUT
END_VAR
IF stURL <> 0 THEN
	__DELETE(stURL				);
END_IF;
IF stKEY <> 0 THEN
	__DELETE(stKEY				);
END_IF;
IF stKEY_ID <> 0 THEN
	__DELETE(stKEY_ID			);
END_IF;
IF stVersion <> 0 THEN
	__DELETE(stVersion			);
END_IF;
IF stResult <> 0 THEN
	__DELETE(stResult			);
END_IF;
IF stTemp <> 0 THEN
	__DELETE(stTemp				);
END_IF;
IF stCommand <> 0 THEN
	__DELETE(stCommand			);
END_IF;
END_METHOD

END_FUNCTION_BLOCK

// 21 Interface/ITF_GRAFANA_LIB_PANEL
INTERFACE ITF_GRAFANA_LIB_PANEL EXTENDS __SYSTEM.IQueryInterface

PROPERTY TABLE_EXECUTE : BOOL
SET
END_SET
GET
END_GET
END_PROPERTY

PROPERTY TABLE_STATUS : STRING
GET
END_GET
END_PROPERTY

PROPERTY LIB_PANEL_UID : STRING
GET
END_GET
END_PROPERTY

END_INTERFACE

// 30 Program Organization Units/fcRemoveSpezialChar
FUNCTION fcRemoveSpezialChar : STRING(255)
VAR_INPUT
	stIn	:	STRING(255);
END_VAR
VAR
	iSafety	:	INT;
	iPos	:	INT;
	iLen	:	INT;
END_VAR

(* Ä *)
iSafety := 0;
WHILE Standard.FIND(stIn,'Ä') <> 0 AND iSafety < 255 DO	
	iPos 		:= Standard.FIND(stIn,'Ä')-1;
	stIn[iPos]	:= 65;	// ANSI A
	stIn[iPos+1]:= 101;	// ANSI e
	iSafety := iSafety + 1;
END_WHILE;
iSafety := 0;
WHILE Standard.FIND(stIn,'ä') <> 0 AND iSafety < 255 DO	
	iPos 		:= Standard.FIND(stIn,'ä')-1;
	stIn[iPos]	:= 97;	// ANSI a
	stIn[iPos+1]:= 101;	// ANSI 3
	iSafety := iSafety + 1;
END_WHILE;
(* Ö *)
iSafety := 0;
WHILE Standard.FIND(stIn,'Ö') <> 0 AND iSafety < 255 DO	
	iPos 		:= Standard.FIND(stIn,'Ö')-1;
	stIn[iPos]	:= 79;	// ANSI O
	stIn[iPos+1]:= 101;	// ANSI e
	iSafety := iSafety + 1;
END_WHILE;
iSafety := 0;
WHILE Standard.FIND(stIn,'ö') <> 0 AND iSafety < 255 DO	
	iPos 		:= Standard.FIND(stIn,'ö')-1;
	stIn[iPos]	:= 111;	// ANSI o
	stIn[iPos+1]:= 101;	// ANSI e
	iSafety := iSafety + 1;
END_WHILE;
(* Ü *)
iSafety := 0;
WHILE Standard.FIND(stIn,'Ü') <> 0 AND iSafety < 255 DO	
	iPos 		:= Standard.FIND(stIn,'Ü')-1;
	stIn[iPos]	:= 85;	// ANSI U
	stIn[iPos+1]:= 101;	// ANSI e
	iSafety := iSafety + 1;
END_WHILE;
iSafety := 0;
WHILE Standard.FIND(stIn,'ü') <> 0 AND iSafety < 255 DO	
	iPos 		:= Standard.FIND(stIn,'ü')-1;
	stIn[iPos]	:= 117;	// ANSI u
	stIn[iPos+1]:= 101;	// ANSI e
	iSafety := iSafety + 1;
END_WHILE;
fcRemoveSpezialChar := stIn;

END_FUNCTION

// 40 Visualizations/VIS_GRAFANA_LIB_PANEL
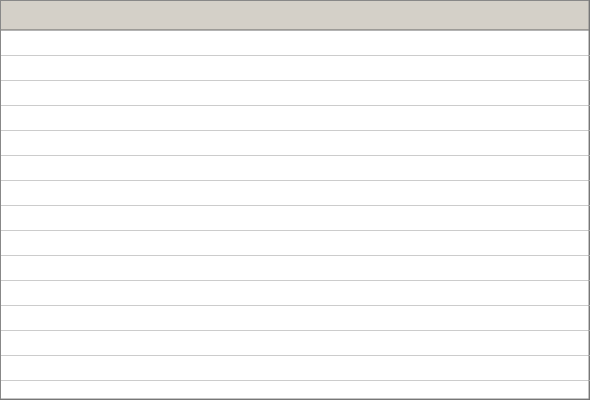
VISUALIZATION VIS_GRAFANA_LIB_PANEL  // 590x400
    Table (0,0 590x400), data array: GVL_GRAFANA_LIB_PANEL.AY_FB_GRAFANA_LIB_PANEL
        p1014161805: Parameter.iMaxLibPanels - 1 + INT#1
        p1128707560: GVL_GRAFANA_LIB_PANEL.iMaxShow
        p3854506369: GVL_GRAFANA_LIB_PANEL.AY_FB_GRAFANA_LIB_PANEL[INDEX].LIB_PANEL_UID
        p1892666644: GVL_GRAFANA_LIB_PANEL.AY_FB_GRAFANA_LIB_PANEL[INDEX].TABLE_EXECUTE
        p338671338: GVL_GRAFANA_LIB_PANEL.AY_FB_GRAFANA_LIB_PANEL[INDEX].TABLE_STATUS
        p2232123230: GRAFANA PANEL ID
        Columns.Column.[1].Template: tap GVL_GRAFANA_LIB_PANEL.AY_FB_GRAFANA_LIB_PANEL[INDEX].TABLE_EXECUTE
END_VISUALIZATION

// 40 Visualizations/VIS_POPUP_GRAFANA
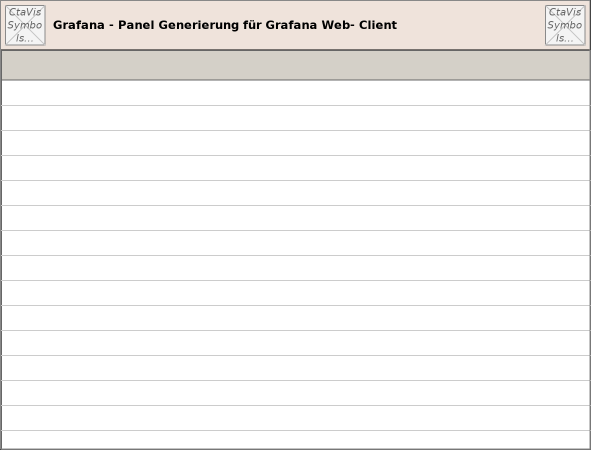
VISUALIZATION VIS_POPUP_GRAFANA  // 591x450
    Rectangle (0,0 591x50)
    Rectangle (0,50 591x400)
    Frame (1,50 590x400)
        shows VIS_GRAFANA_LIB_PANEL()
    Image (5,5 40x40), image: CtaVisSymbols.ImagePool.Grafana_Logo
    Image (545,5 40x40), image: CtaVisSymbols.ImagePool.close_solo_black
        OnMouseClick:  Dialog=VIS_POPUP_GRAFANA, Result=None, NumpadKeypadSet=True
    Label (50,15 500x20), "Grafana - Panel Generierung für Grafana Web- Client"
END_VISUALIZATION
